(*

.. <legal notes>

legal notes
=================
| SPDX-FileCopyrightText: © 2026 Oleksandr Tiutyk <trofimich@gmail.com>
| SPDX-License-Identifier: LGPL-3.0-only
| For details check: LGPL-3.0-only_

.. _LGPL-3.0-only: https://www.gnu.org/licenses/lgpl-3.0.en.html

.. </legal notes>

*)

FUNCTION_BLOCK ABSTRACT CompositeDevice
VAR_GENERIC CONSTANT
    _SubDeviceCount : INT(0..1000) := 0;
END_VAR
EXTENDS Device IMPLEMENTS IInputDevice, IOutputDevice

METHOD FINAL Disable
VAR
	i : INT;
END_VAR
IF _Enabled THEN
	OnEnabledChanging(FALSE);
END_IF

IF __ISVALIDREF(SubDevices) AND_THEN _SubDeviceCount > 0 THEN
	FOR i := 0 TO _SubDeviceCount - 1 DO
		SubDevices[i].Disable();
	END_FOR	
END_IF

IF _Enabled THEN
	_Enabled := FALSE;
	
	OnEnabledChanged();
END_IF
END_METHOD

METHOD FINAL Enable
VAR_INPUT
	includeChildren : BOOL := TRUE;
END_VAR
VAR
	i : INT;
END_VAR
IF NOT _Enabled THEN
	OnEnabledChanging(TRUE);
END_IF

IF __ISVALIDREF(SubDevices) AND_THEN _SubDeviceCount > 0 THEN
	FOR i := 0 TO _SubDeviceCount - 1 DO
		SubDevices[i].Enable();
	END_FOR	
END_IF

IF NOT _Enabled THEN
	_Enabled := TRUE;
	
	OnEnabledChanged();
END_IF

Parent.Enable(FALSE);
END_METHOD

METHOD FINAL Initialize : BOOL
VAR
	i : INT;
	
	memberNotSpecifiedException : Core.DataMemberNotSpecifiedException;	
END_VAR
IF _Parent = 0 THEN
	memberNotSpecifiedException.Throw(Namespacename, ClassName, __POUNAME(), __POSITION(), 'Parent');
END_IF

IF _SubDeviceCount > 0 AND_THEN NOT __ISVALIDREF(SubDevices) THEN
	memberNotSpecifiedException.Throw(Namespacename, ClassName, __POUNAME(), __POSITION(), 'SubDevices');
END_IF

OnPreSubDeviceInitializing();

Initialize := TRUE;

IF _SubDeviceCount > 0 THEN
	FOR i := 0 TO _SubDeviceCount - 1 DO
		IF SubDevices[i] = 0 THEN
			memberNotSpecifiedException.Throw(Namespacename, ClassName, __POUNAME(), __POSITION(), Core.Strings.Concat255('SubDevices[', TO_STRING(i), ']'));						
		END_IF
		
		Initialize := Initialize AND SubDevices[i].Initialize();
	END_FOR
END_IF

Initialize := OnPostSubDeviceInitializing();
END_METHOD

METHOD PROTECTED OnEnabledChanged
END_METHOD

METHOD PROTECTED OnEnabledChanging 
VAR_INPUT
	newValue : BOOL;
END_VAR
END_METHOD

METHOD PROTECTED OnInputProcessed
END_METHOD

METHOD PROTECTED OnInputProcessing
END_METHOD

METHOD PROTECTED OnOutputProcessed
END_METHOD

METHOD PROTECTED OnOutputProcessing
END_METHOD

METHOD PROTECTED OnPostSubDeviceInitializing : BOOL
OnPostSubDeviceInitializing := TRUE;
END_METHOD

METHOD PROTECTED OnPreSubDeviceInitializing
END_METHOD

METHOD FINAL ProcessInput
VAR
	i : INT;
	
	inputSubDevice : IInputDevice;
END_VAR
OnInputProcessing();

IF __ISVALIDREF(SubDevices) AND_THEN _SubDeviceCount > 0 THEN
	FOR i := 0 TO _SubDeviceCount - 1 DO
		IF NOT SubDevices[i].Enabled OR_ELSE NOT __QUERYINTERFACE(SubDevices[i], inputSubDevice) THEN
			CONTINUE;
		END_IF
		
		inputSubDevice.ProcessInput();
	END_FOR	
END_IF

OnInputProcessed();
END_METHOD

METHOD FINAL ProcessOutput
VAR
	i : INT;
	
	outputSubDevice : IOutputDevice;
END_VAR
OnOutputProcessing();

IF __ISVALIDREF(SubDevices) AND_THEN _SubDeviceCount > 0 THEN
	FOR i := 0 TO _SubDeviceCount - 1 DO
		IF NOT SubDevices[i].Enabled OR_ELSE NOT __QUERYINTERFACE(SubDevices[i], outputSubDevice) THEN
			CONTINUE;
		END_IF
		
		outputSubDevice.ProcessOutput();
	END_FOR	
END_IF

OnOutputProcessed();
END_METHOD

{attribute 'monitoring' := 'call'}
PROPERTY FINAL SubDeviceCount : INT
GET
SubDeviceCount := _SubDeviceCount;
END_GET
END_PROPERTY

{attribute 'monitoring' := 'call'}
PROPERTY ABSTRACT SubDevices : REFERENCE TO ARRAY [0.._SubDeviceCount - 1] OF IDevice
GET
END_GET
END_PROPERTY

METHOD FINAL TryGetSubDeviceByIndex : IDevice
VAR_INPUT
	index : BYTE;
END_VAR
IF index < 0 OR_ELSE index >= _SubDeviceCount OR_ELSE NOT __ISVALIDREF(SubDevices) THEN
	RETURN;
END_IF

TryGetSubDeviceByIndex := SubDevices[index];
END_METHOD

END_FUNCTION_BLOCK

(* stored: Version 1.1.0.1
   POU CompositeDevice: Id {25bfda0d-9225-4be2-8314-f8314e830df8}, SpecialFunc None
   Folder Internal members to override: Id {7fd0c34a-cb46-4c3c-b337-f69fec474a23}
   Folder EnabledChange: Id {e7fb94cc-52bc-4813-ac3d-f0ccfefbf254}
   Folder Initialization: Id {0d65471c-cd65-4df9-bf5f-c01d4ef54625}
   Folder ProcessInput: Id {79809b58-7d71-4b75-b242-a4aba637ef2e}
   Folder ProcessOutput: Id {9f8de15a-1166-4374-8d27-0103e613ff6e}
   Method Disable: Id {53188197-be8e-4525-aeae-812ec12422bf}
   Method Enable: Id {6182586a-d1b9-4b36-ba6f-359d49e6858f}
   Method Initialize: Id {39df2100-ad47-414a-b2a1-58201a8bb85e}
   Method OnEnabledChanged: Id {72495f3a-cbb8-41b2-b62b-87df10ab8ca7}
   Method OnEnabledChanging: Id {b83d234d-f0de-4bbb-a430-648c37cbe155}
   Method OnInputProcessed: Id {f3d4720d-fb6f-4ac6-b198-9c6a9d344a6d}
   Method OnInputProcessing: Id {0d78f97b-abdf-4c22-b28b-d5acc1dd05d9}
   Method OnOutputProcessed: Id {6dafed43-c189-43e6-b75c-e7d4c90c0264}
   Method OnOutputProcessing: Id {b6627520-7954-4ce0-bc86-cc49fe1d6ac6}
   Method OnPostSubDeviceInitializing: Id {92cef328-43a3-40eb-82aa-0ebd1e9574ce}
   Method OnPreSubDeviceInitializing: Id {5981974c-d168-46b8-b69e-2cfb74c40a1a}
   Method ProcessInput: Id {169f608c-73af-42d0-b266-fd32baea3032}
   Method ProcessOutput: Id {d8822de7-f12d-43fe-bdcd-3812e5246f80}
   Property SubDeviceCount: Id {8fe9b9a1-849f-40ca-953d-31f713106361}
   Get Get: Id {efd6679f-7abb-4ba2-907a-97a3a87b2c0a}
   Property SubDevices: Id {5eb8cc14-af21-41a6-964e-854d2107c6da}
   Get Get: Id {92c9163e-e171-4a3b-8e8e-5251e6af78eb}
   Method TryGetSubDeviceByIndex: Id {e2e78db3-9f06-4b18-b030-d1b97840dae7} *)
